INTERFACE I_AxisEnable EXTENDS I_Enablable, I_Override

{attribute 'monitoring' := 'call'}
PROPERTY InhibitFeedBackward : BOOL
GET
END_GET
SET
END_SET
END_PROPERTY

{attribute 'monitoring' := 'call'}
PROPERTY InhibitFeedForward : BOOL
GET
END_GET
SET
END_SET
END_PROPERTY

END_INTERFACE

(* stored: Version 1.1.0.1, ProductVersion 3.1.4026.18
   Itf I_AxisEnable: Id {73aa81ef-0a82-4a2d-aafa-259a7a2e1a2b}
   Property InhibitFeedBackward: Id {f78063d2-25c6-4eb4-8d5b-65b6b29beef9}
   Get Get: Id {7c7a5b76-2daa-4457-8e22-71a2d8b1daaa}
   Set Set: Id {1dfd0723-275b-4bc3-91bb-eda4def07f23}
   Property InhibitFeedForward: Id {87ba04a3-84a0-42af-9c04-cf0266b258df}
   Get Get: Id {26d69f0b-ec61-480f-9b86-14ec9c24633d}
   Set Set: Id {c6e71f21-8f66-47d9-9a42-5f83b6c8c59e} *)
